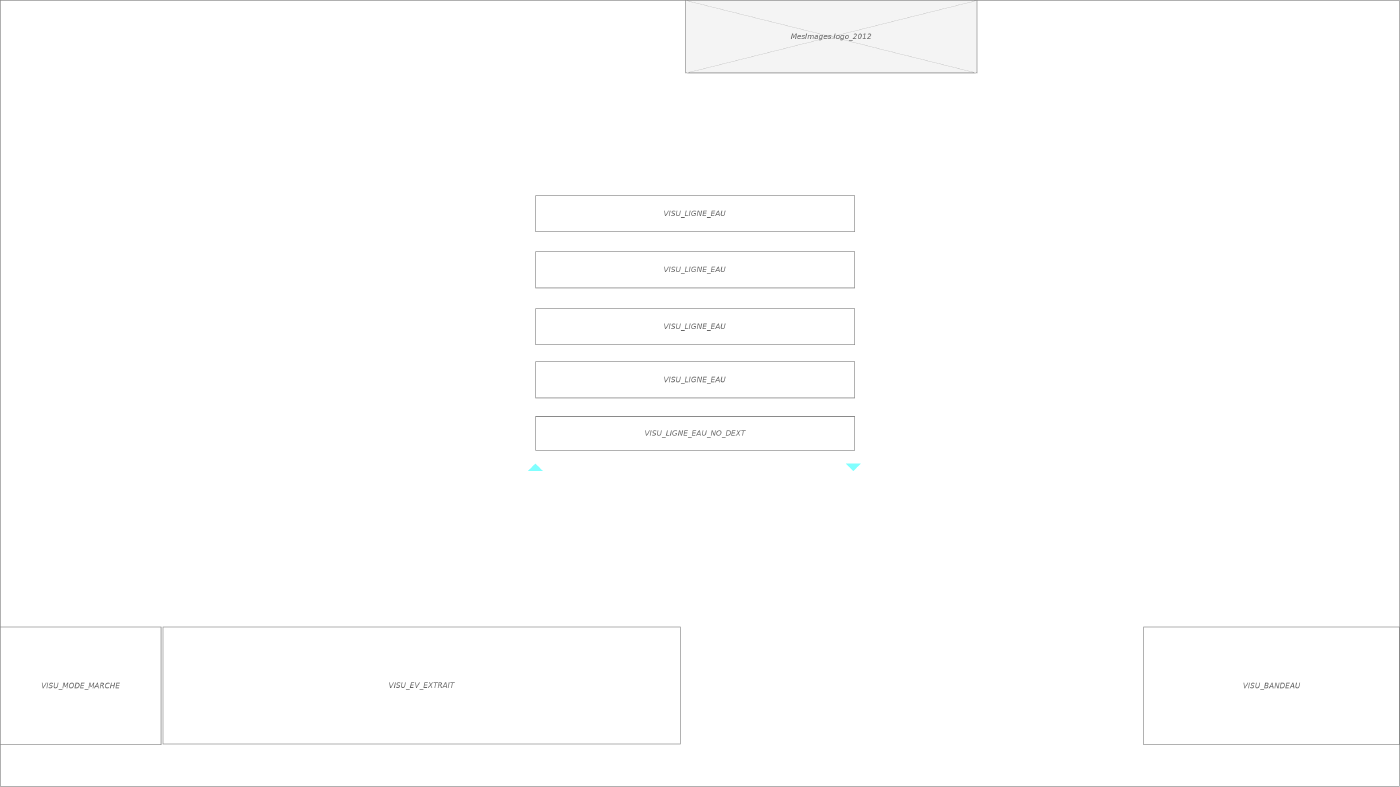
VISUALIZATION SYN_SERVITUDES  // 1920x1080, background image fond_blanc_1280_1024
    Frame (223,860 710x161)
        shows VISU_EV_EXTRAIT()
    Frame (1568,860 352x162)
        shows VISU_BANDEAU(m_Input_MACHINE := Global_Variables.MACHINE)
    Frame (0,860 221x162)
        shows VISU_MODE_MARCHE(m_Input_MACHINE := .MACHINE)
    Polyline (403,450)
    Polyline (403,450)
    Polygon (734,636) (724,646) (744,646)
    Polygon (1170,646) (1160,636) (1180,636)
    Image (940,0 400x100), image: MesImages.logo_2012
    Frame (734,496 438x50)
        shows VISU_LIGNE_EAU(m_Input_LIGNE_EAU := PRG_SERVITUDES.LIGNE_REF[4])
    Frame (734,571 438x47)
        shows VISU_LIGNE_EAU_NO_DEXT(m_Input_LIGNE_EAU := PRG_SERVITUDES.LIGNE_REF[5])
    Frame (734,268 438x50)
        shows VISU_LIGNE_EAU(m_Input_LIGNE_EAU := PRG_SERVITUDES.LIGNE_REF[1])
    Frame (734,345 438x50)
        shows VISU_LIGNE_EAU(m_Input_LIGNE_EAU := PRG_SERVITUDES.LIGNE_REF[2])
    Frame (734,423 438x50)
        shows VISU_LIGNE_EAU(m_Input_LIGNE_EAU := PRG_SERVITUDES.LIGNE_REF[3])
END_VISUALIZATION

(* stored: Version 1.1.0.1, ProductVersion 3.1.4026.18
   Visu SYN_SERVITUDES: Id {b3c614b1-82a8-47d3-8c47-9b50ae71f55f} *)
